Staubli VAL3: getVersion.pgx

public program getVersion(string& x_sVersion[] (dimensions=1))
begin
  // This program returns the version number of the library
  //
  // Input Param
  //  none       :
  //
  // Output param
  //  x_sVersion  : Software version
  //
  //----------------------------------------------------------------
  //
  x_sVersion=cfg:sVERSION
end
